FUNCTION_BLOCK FB_WorkerDefGrid_Verify EXTENDS FB_WorkerDefGrid
VAR_OUTPUT
  bWateGateActive   AT%Q* : BOOL;     //  wate gate activation pulse
END_VAR
VAR
  lastEjected   : BOOL;   // stores state if last CT was ejected 
  tpEjectPulse  : TP := (PT:=T#100MS);
  
  // print manager reference
  _pPm : POINTER TO FB_Pm_DMAX;
END_VAR
VAR PERSISTENT
  _fWorkerToPu   : LREAL := 1.2;    (*Distance between PU and this worker, mechanisch*)
END_VAR

METHOD PROTECTED  Attach : BOOL
VAR_INPUT
  iCT              : I_CT;                         (*container at triggered event position*)
END_VAR
VAR 
  bSuccess         : BOOL;
END_VAR
IF SUPER^.Attach(iCT:=iCT) THEN
  
  // do CT supervision here and decice what happens with this sheet
   bSuccess := TRUE;
  IF NOT iCT.bValid AND iCT.bProductPresent AND iCT.pJob <> 0 THEN
    bSuccess := FALSE;
    // tag for ejection
    iCT.pCT^.lPrOutput := EN_PrinterOutput.trash;
	END_IF

  // finish CT in production
  IF _pPm <> 0 THEN 
    _pPm^.CT_Finish(sCT:=iCT, bSuccess:=bSuccess);
  ELSE
    LogError('PrintManager not set');
	END_IF
  
  // select output
  IF iCT.pCT^.lPrOutput = EN_PrinterOutput.trash THEN
    // create eject trigger
    tpEjectPulse(IN:=TRUE);
    lastEjected := TRUE;
  ELSE
    tpEjectPulse(IN:=FALSE);
    lastEjected := FALSE;
	END_IF
  
END_IF
END_METHOD

PROPERTY fWorkerToPu : LREAL
GET
fWorkerToPu := _fWorkerToPu;
END_GET
END_PROPERTY

METHOD   mJobStart
VAR_INPUT
	sJobDef	: CalmarCompPrint.I_JobDefinition;
END_VAR

_bJobActive := TRUE;
END_METHOD

METHOD  mJobStop
VAR_INPUT
	sStatus	: CalmarCompPrint.I_JobStatus;
END_VAR
_bJobActive := FALSE;
END_METHOD

METHOD Release : BOOL
VAR_INPUT
  iCT              : I_CT;                         (*container at triggered event position*)
END_VAR
IF SUPER^.Release(iCT := iCT) THEN
  ;
END_IF
END_METHOD

(*
  Set PrintManager.
*)
METHOD setPm : BOOL
VAR_INPUT
  pPm : POINTER TO FB_Pm_DMAX;
END_VAR
IF pPm = 0 THEN LogError('Invalid Pm given'); END_IF

_pPm := pPm;  // register print manager reference
END_METHOD

METHOD  work
VAR_INST
  fT_Pulse  : F_TRIG;
END_VAR
SUPER^.work();

//Worker position update
IF _pParamMediator <> 0 AND _pAttachedCt = 0 THEN     // Update only without attached container
  // WorkerPosition =  Worker<-PU<-CAM<-SheetDetect
  fPosition := _fWorkerToPu + _pParamMediator^.fCameraToPrintOffset + _pParamMediator^.fDetectToCamera;
END_IF

IF _pAttachedCt <> 0 THEN
  tpEjectPulse(Q=>bWateGateActive);
  fT_Pulse(CLK:=bWateGateActive);
  
  // release
  IF tpEjectPulse.IN THEN
    IF fT_Pulse.Q THEN  
      tpEjectPulse(IN:=FALSE);
      LogLvl(Lvl:=E_LogSeverity.Debug, Msg:=F_Concat2('Eject CT: ', _pAttachedCt^.print(0)));
      Release(iCT:=_pAttachedCt^);
    END_IF
  ELSE
    Release(iCT:=_pAttachedCt^);
  END_IF
END_IF
END_METHOD

END_FUNCTION_BLOCK

(* stored: Version 1.1.0.1, ProductVersion 3.1.4024.3
   POU FB_WorkerDefGrid_Verify: Id {ba30a803-cb22-4c70-92de-a30f80d703f5}, SpecialFunc None
   Method Attach: Id {ed09302e-2885-443a-873e-e5493c07daba}
   Property fWorkerToPu: Id {d213abe5-dfd5-4330-9682-099f2ba8982a}
   Get Get: Id {530a8023-6b19-4384-9a2f-e3a75c3159cc}
   Method mJobStart: Id {4a0a5887-5c40-49ea-8411-5fb79e221249}
   Method mJobStop: Id {d134956b-60c5-4e97-96a0-a8378694c410}
   Method Release: Id {c5bbf20b-0ff6-499b-bfe5-090aa809106f}
   Method setPm: Id {b89f6ac4-9ac9-4bfe-8bb7-e25e99bfe006}
   Method work: Id {f3293130-827d-4f71-beb2-d681c617967b} *)
